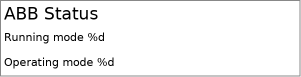
VISUALIZATION _VisuABBStatus  // 301x77
    Label (1,1 148x25), "ABB Status"
    Rectangle (1,25 298x25), "Running mode %d", text variable: ComGVL._gABBRunTable[ComGVL._fbTryOutABBRunMode ]
    Rectangle (1,50 298x25), "Operating mode %d", text variable: ComGVL._gABBOpTable[ComGVL._fbTryOutABBOpMode ]
END_VISUALIZATION

(* stored: Version 1.1.0.1, ProductVersion 3.1.4024.2
   Visu _VisuABBStatus: Id {3493fc79-3a22-4550-9216-cb05317ffb73} *)
